FUNCTION_BLOCK EL3114
VAR
	_io : EL3xx4_Data;
	{attribute addProperty Name "WcState"}
	_wcState : WcStateInputToggle;
	{attribute addProperty Name "Info data"}
	_infoData : InfoDataAds;
END_VAR

PROPERTY IO : REFERENCE TO EL3xx4_Data
GET
IO REF= _io;
END_GET
END_PROPERTY

PROPERTY WcState : REFERENCE TO WcStateInputToggle
GET
WcState REF= _wcState;
END_GET
END_PROPERTY

END_FUNCTION_BLOCK

(* stored: Version 1.1.0.1, ProductVersion 3.1.4024.9
   POU EL3114: Id {14296822-9ec7-0c0a-1699-71e74cb6a597}, SpecialFunc None
   Property IO: Id {475ce373-5bc5-08c6-12fa-247bdd2e705f}
   Get Get: Id {065c1711-d2c1-0020-2645-bdf5ab6be078}
   Property WcState: Id {168975b4-c6b0-0b2f-33e7-ea0af4322d36}
   Get Get: Id {b7d72852-0b26-0941-2fd8-55f9a0cef47d} *)
